FUNCTION_BLOCK E_CYCLE (* Peroidic event generator *)
  (* Standard: 61499-1 Annex A; Description: Copyright (c) 2017 fortiss GmbH This program and the accompanying materials are made available under the terms of the Eclipse Public License 2.0 which is available at https://www.eclipse.org/legal/epl-2.0/ SPDX-License-Identifier: EPL-2.0 *)
  (* Version 1.0, 2017-09-21, Alois Zoitl, fortiss GmbH, initial API and implementation and/or initial documentation *)
  (* Version 3.0, 2025-04-14, Patrick Aigner, changed package *)
  PACKAGE iec61499::events;
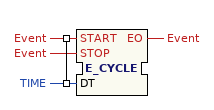
  EVENT_INPUT
    START WITH DT; (* Start the perodic generation of events *)
    STOP; (* Stop the generation of events *)
  END_EVENT
  EVENT_OUTPUT
    EO; (* Periodically triggered output event *)
  END_EVENT
  VAR_INPUT
    DT : TIME; (* cycle time *)
  END_VAR
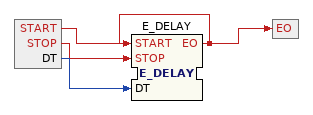
  FBS
    E_DELAY : iec61499::events::E_DELAY;
  END_FBS
  EVENT_CONNECTIONS
    START TO E_DELAY.START;
    STOP TO E_DELAY.STOP;
    E_DELAY.EO TO E_DELAY.START;
    E_DELAY.EO TO EO;
  END_CONNECTIONS
  DATA_CONNECTIONS
    DT TO E_DELAY.DT;
  END_CONNECTIONS
END_FUNCTION_BLOCK
